(*
Checks if two traffic phases are compatible using their phase identity number.
Two compatible traffic phases can be run concurrently without causing traffic
conflicts.
*)

FUNCTION Check_Phase_Compatibility : Bool
VAR_INPUT
	fb_Phase_A : REFERENCE TO fb_Traffic_Phase;
	fb_Phase_B : REFERENCE TO fb_Traffic_Phase;
END_VAR
VAR
	n_ID_A : UINT := fb_Phase_A.st_Phase_Info.n_Phase_Identity;
	n_ID_B : UINT := fb_Phase_B.st_Phase_Info.n_Phase_Identity;
END_VAR

// Check the street identity
IF fb_Phase_A.st_Phase_Info.e_Street_Identity = fb_Phase_B.st_Phase_Info.e_Street_Identity THEN
	// Check if one ID is odd and one is even
	IF (n_ID_A + n_ID_B) MOD 2 = 1 THEN
		// If the phase numbers add to 7, meaning we have a 1 + 6 or 2 + 5 pair for the major street
		// or if the phase numbers add to 11, meaning we have a 3 + 8 or 4 + 7 pair for the minor street
		IF (n_ID_A + n_ID_B) = 7 OR (n_ID_A + n_ID_B) = 11 THEN
			Check_Phase_Compatibility := TRUE;
			
		// Other possible configurations are incompatible
		ELSE
			Check_Phase_Compatibility := FALSE;
		END_IF
	
	// IDs are either both odd or both even
	ELSE
		Check_Phase_Compatibility := TRUE;
	END_IF

ELSE
	Check_Phase_Compatibility := FALSE;
END_IF

END_FUNCTION

(* stored: Version 1.1.0.1
   POU Check_Phase_Compatibility: Id {d35923ca-f9be-4f8a-b919-3bef0a4502e7}, SpecialFunc None *)
